TYPE ACRMemoryTimeEvent EXTENDS ACRMemoryEvent :
STRUCT
		_Value : TIME;
END_STRUCT
END_TYPE

(* stored: Version 1.1.0.1, ProductVersion 3.1.4020.12
   DUT ACRMemoryTimeEvent: Id {4bea79bc-4267-41c9-8646-53972a082031} *)
